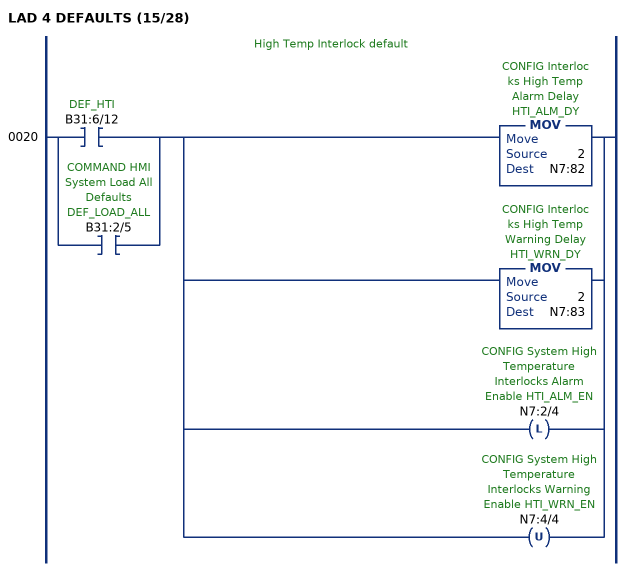
% Rung: 20 %
% High Temp Interlock default %
SOR BST XIC B31:6/12 NXB XIC B31:2/5 BND BST MOV 2 N7:82 NXB MOV 2 N7:83 NXB OTL N7:2/4 NXB OTU N7:4/4 BND EOR
%   B31:6/12  DEF_HTI %
%   B31:2/5  DEF_LOAD_ALL  "COMMAND HMI System Load All Defaults" %
%   N7:82  HTI_ALM_DY  "CONFIG Interlocks High Temp Alarm Delay" %
%   N7:83  HTI_WRN_DY  "CONFIG Interlocks High Temp Warning Delay" %
%   N7:2/4  HTI_ALM_EN  "CONFIG System High Temperature Interlocks Alarm Enable" %
%   N7:4/4  HTI_WRN_EN  "CONFIG System High Temperature Interlocks Warning Enable" %

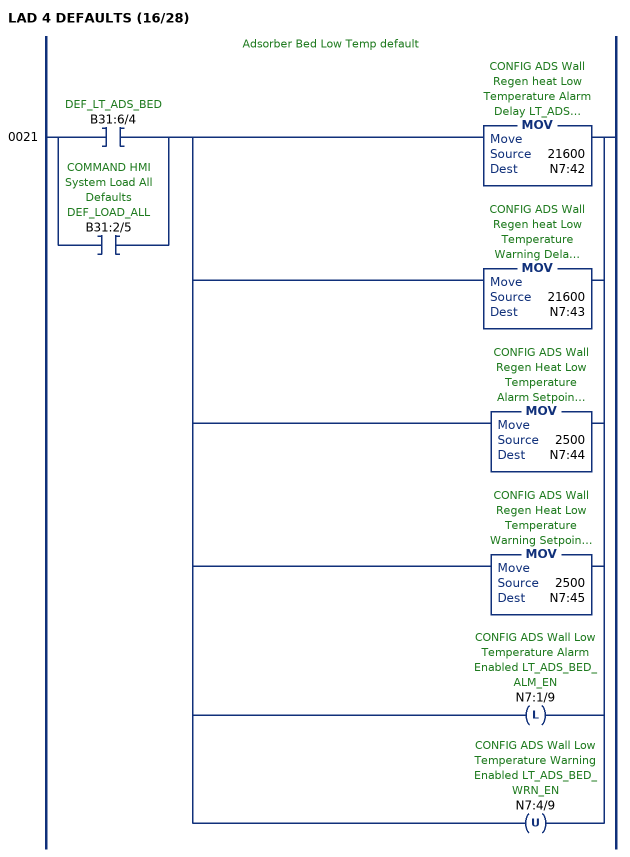
% Rung: 21 %
% Adsorber Bed Low Temp default %
SOR BST XIC B31:6/4 NXB XIC B31:2/5 BND BST MOV 21600 N7:42 NXB MOV 21600 N7:43 NXB MOV 2500 N7:44 NXB MOV 2500 N7:45 NXB OTL N7:1/9 NXB OTU N7:4/9 BND EOR
%   B31:6/4  DEF_LT_ADS_BED %
%   B31:2/5  DEF_LOAD_ALL  "COMMAND HMI System Load All Defaults" %
%   N7:42  LT_ADS_BED_ALM_DLY  "CONFIG ADS Wall Regen heat Low Temperature Alarm Delay" %
%   N7:43  LT_ADS_BED_WRN_DLY  "CONFIG ADS Wall Regen heat Low Temperature Warning Delay" %
%   N7:44  LT_ADS_BED_ALM_SP  "CONFIG ADS Wall Regen Heat Low Temperature Alarm Setpoint" %
%   N7:45  LT_ADS_BED_WRN_SP  "CONFIG ADS Wall Regen Heat Low Temperature Warning Setpoint" %
%   N7:1/9  LT_ADS_BED_ALM_EN  "CONFIG ADS Wall Low Temperature Alarm Enabled" %
%   N7:4/9  LT_ADS_BED_WRN_EN  "CONFIG ADS Wall Low Temperature Warning Enabled" %

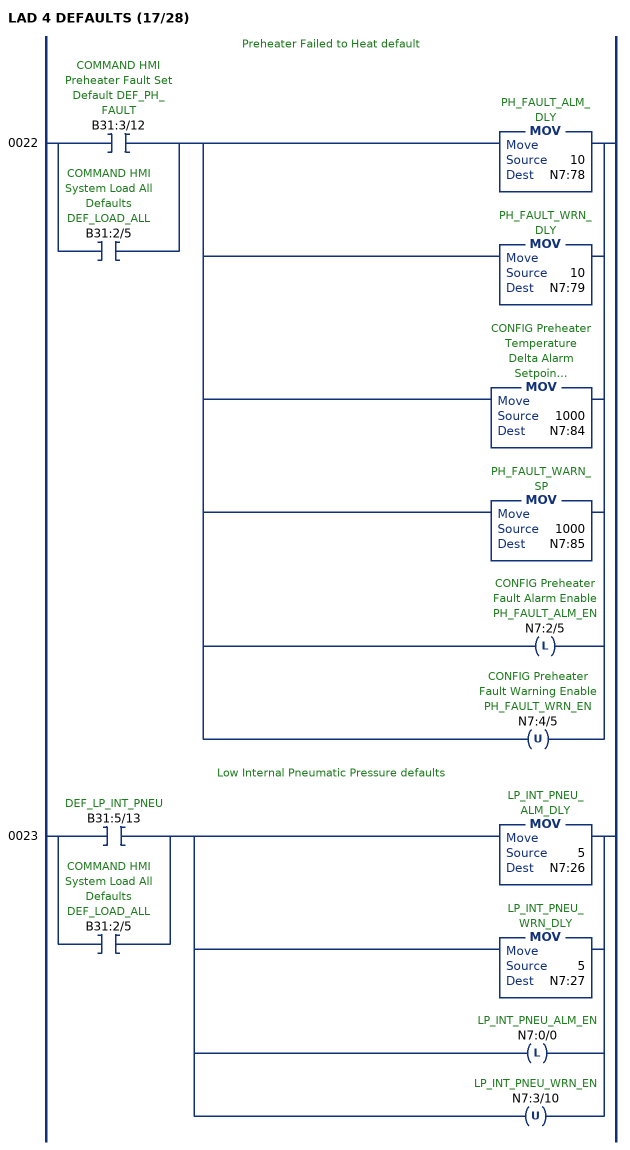
% Rung: 22 %
% Preheater Failed to Heat default %
SOR BST XIC B31:3/12 NXB XIC B31:2/5 BND BST MOV 10 N7:78 NXB MOV 10 N7:79 NXB MOV 1000 N7:84 NXB MOV 1000 N7:85 NXB OTL N7:2/5 NXB OTU N7:4/5 BND EOR
%   B31:3/12  DEF_PH_FAULT  "COMMAND HMI Preheater Fault Set Default" %
%   B31:2/5  DEF_LOAD_ALL  "COMMAND HMI System Load All Defaults" %
%   N7:78  PH_FAULT_ALM_DLY %
%   N7:79  PH_FAULT_WRN_DLY %
%   N7:84  PH_FAULT_ALARM_SP  "CONFIG Preheater Temperature Delta Alarm Setpoint" %
%   N7:85  PH_FAULT_WARN_SP %
%   N7:2/5  PH_FAULT_ALM_EN  "CONFIG Preheater Fault Alarm Enable" %
%   N7:4/5  PH_FAULT_WRN_EN  "CONFIG Preheater Fault Warning Enable" %
% Rung: 23 %
% Low Internal Pneumatic Pressure defaults %
SOR BST XIC B31:5/13 NXB XIC B31:2/5 BND BST MOV 5 N7:26 NXB MOV 5 N7:27 NXB OTL N7:0/0 NXB OTU N7:3/10 BND EOR
%   B31:5/13  DEF_LP_INT_PNEU %
%   B31:2/5  DEF_LOAD_ALL  "COMMAND HMI System Load All Defaults" %
%   N7:26  LP_INT_PNEU_ALM_DLY %
%   N7:27  LP_INT_PNEU_WRN_DLY %
%   N7:0/0  LP_INT_PNEU_ALM_EN %
%   N7:3/10  LP_INT_PNEU_WRN_EN %

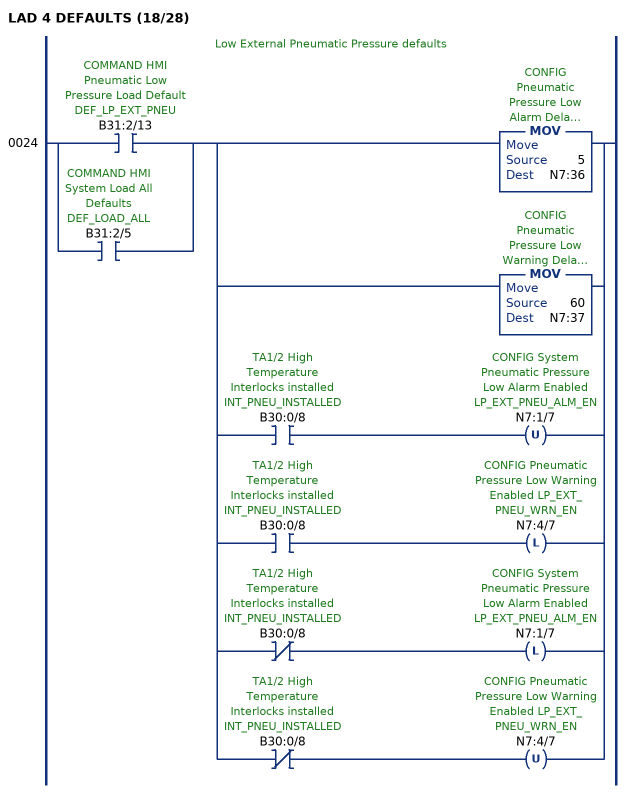
% Rung: 24 %
% Low External Pneumatic Pressure defaults %
SOR BST XIC B31:2/13 NXB XIC B31:2/5 BND BST MOV 5 N7:36 NXB MOV 60 N7:37 NXB XIC B30:0/8 OTU N7:1/7 NXB XIC B30:0/8 OTL N7:4/7 NXB XIO B30:0/8 OTL N7:1/7 NXB XIO B30:0/8 OTU N7:4/7 BND EOR
%   B31:2/13  DEF_LP_EXT_PNEU  "COMMAND HMI Pneumatic Low Pressure Load Default" %
%   B31:2/5  DEF_LOAD_ALL  "COMMAND HMI System Load All Defaults" %
%   N7:36  LP_EXT_PNEU_ALM_DLY  "CONFIG Pneumatic Pressure Low Alarm Delay" %
%   N7:37  LP_EXT_PNEU_WRN_DLY  "CONFIG Pneumatic Pressure Low Warning Delay" %
%   B30:0/8  INT_PNEU_INSTALLED  "TA1/2 High Temperature Interlocks installed" %
%   N7:1/7  LP_EXT_PNEU_ALM_EN  "CONFIG System Pneumatic Pressure Low Alarm Enabled" %
%   N7:4/7  LP_EXT_PNEU_WRN_EN  "CONFIG Pneumatic Pressure Low Warning Enabled" %

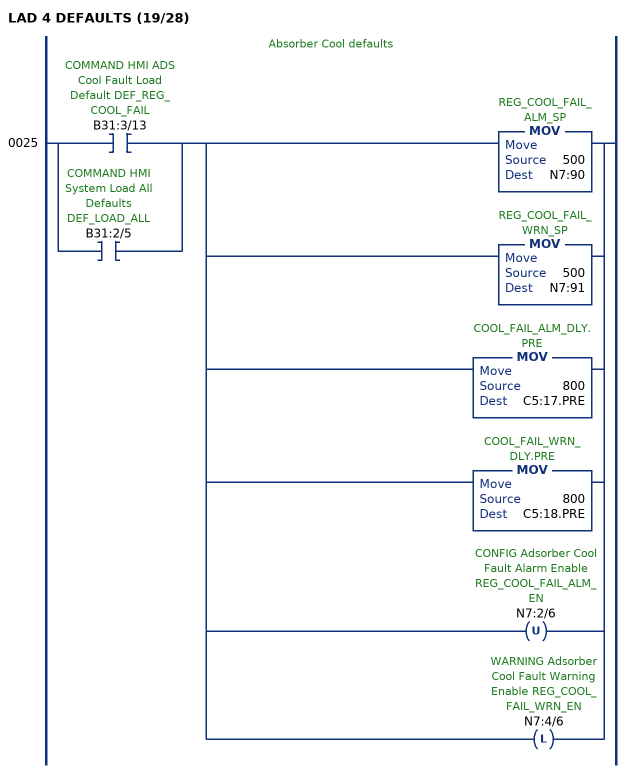
% Rung: 25 %
% Absorber Cool defaults %
SOR BST XIC B31:3/13 NXB XIC B31:2/5 BND BST MOV 500 N7:90 NXB MOV 500 N7:91 NXB MOV 800 C5:17.PRE NXB MOV 800 C5:18.PRE NXB OTU N7:2/6 NXB OTL N7:4/6 BND EOR
%   B31:3/13  DEF_REG_COOL_FAIL  "COMMAND HMI ADS Cool Fault Load Default" %
%   B31:2/5  DEF_LOAD_ALL  "COMMAND HMI System Load All Defaults" %
%   N7:90  REG_COOL_FAIL_ALM_SP %
%   N7:91  REG_COOL_FAIL_WRN_SP %
%   C5:17  COOL_FAIL_ALM_DLY %
%   C5:18  COOL_FAIL_WRN_DLY %
%   N7:2/6  REG_COOL_FAIL_ALM_EN  "CONFIG Adsorber Cool Fault Alarm Enable" %
%   N7:4/6  REG_COOL_FAIL_WRN_EN  "WARNING Adsorber Cool Fault Warning Enable" %

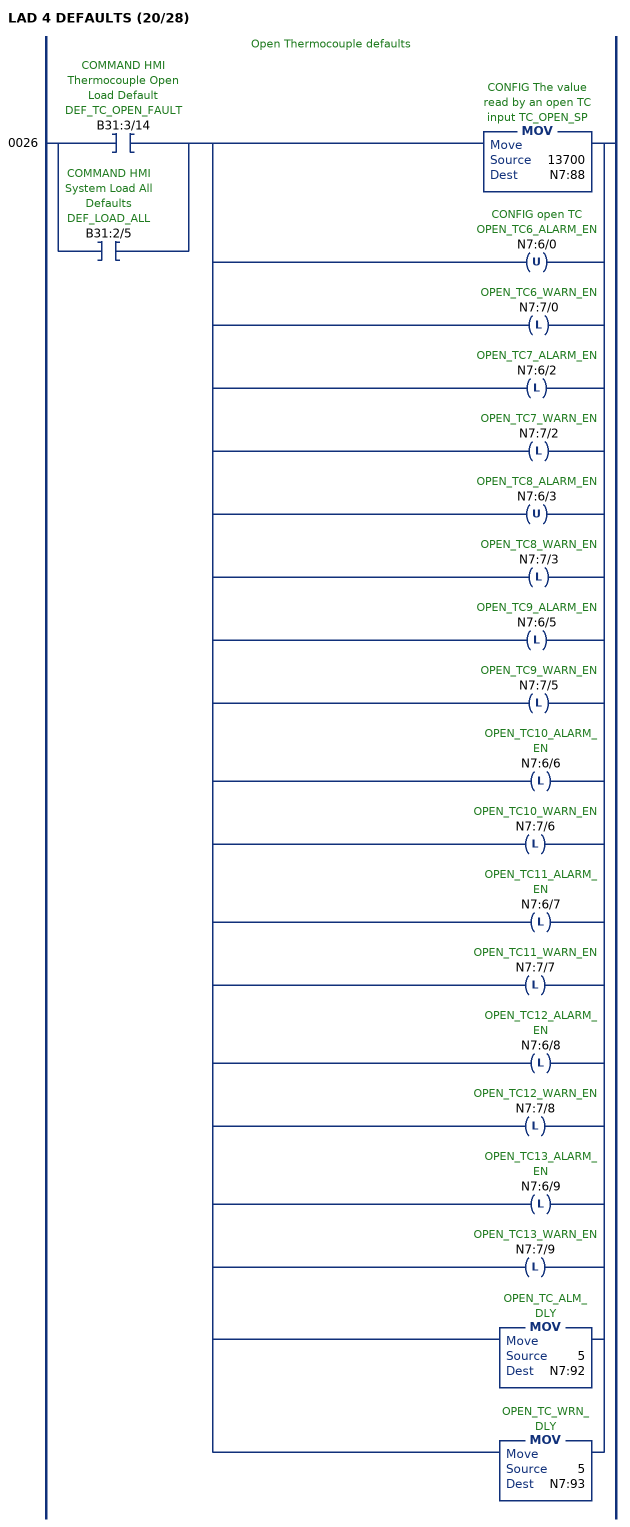
% Rung: 26 %
% Open Thermocouple defaults %
SOR BST XIC B31:3/14 NXB XIC B31:2/5 BND BST MOV 13700 N7:88 NXB OTU N7:6/0 NXB OTL N7:7/0 NXB OTL N7:6/2 NXB OTL N7:7/2 NXB OTU N7:6/3 NXB OTL N7:7/3 NXB OTL N7:6/5 NXB OTL N7:7/5 NXB OTL N7:6/6 NXB OTL N7:7/6 NXB OTL N7:6/7 NXB OTL N7:7/7 NXB OTL N7:6/8 NXB OTL N7:7/8 NXB OTL N7:6/9 NXB OTL N7:7/9 NXB MOV 5 N7:92 NXB MOV 5 N7:93 BND EOR
%   B31:3/14  DEF_TC_OPEN_FAULT  "COMMAND HMI Thermocouple Open Load Default" %
%   B31:2/5  DEF_LOAD_ALL  "COMMAND HMI System Load All Defaults" %
%   N7:88  TC_OPEN_SP  "CONFIG The value read by an open TC input" %
%   N7:6/0  OPEN_TC6_ALARM_EN  "CONFIG open TC" %
%   N7:7/0  OPEN_TC6_WARN_EN %
%   N7:6/2  OPEN_TC7_ALARM_EN %
%   N7:7/2  OPEN_TC7_WARN_EN %
%   N7:6/3  OPEN_TC8_ALARM_EN %
%   N7:7/3  OPEN_TC8_WARN_EN %
%   N7:6/5  OPEN_TC9_ALARM_EN %
%   N7:7/5  OPEN_TC9_WARN_EN %
%   N7:6/6  OPEN_TC10_ALARM_EN %
%   N7:7/6  OPEN_TC10_WARN_EN %
%   N7:6/7  OPEN_TC11_ALARM_EN %
%   N7:7/7  OPEN_TC11_WARN_EN %
%   N7:6/8  OPEN_TC12_ALARM_EN %
%   N7:7/8  OPEN_TC12_WARN_EN %
%   N7:6/9  OPEN_TC13_ALARM_EN %
%   N7:7/9  OPEN_TC13_WARN_EN %
%   N7:92  OPEN_TC_ALM_DLY %
%   N7:93  OPEN_TC_WRN_DLY %

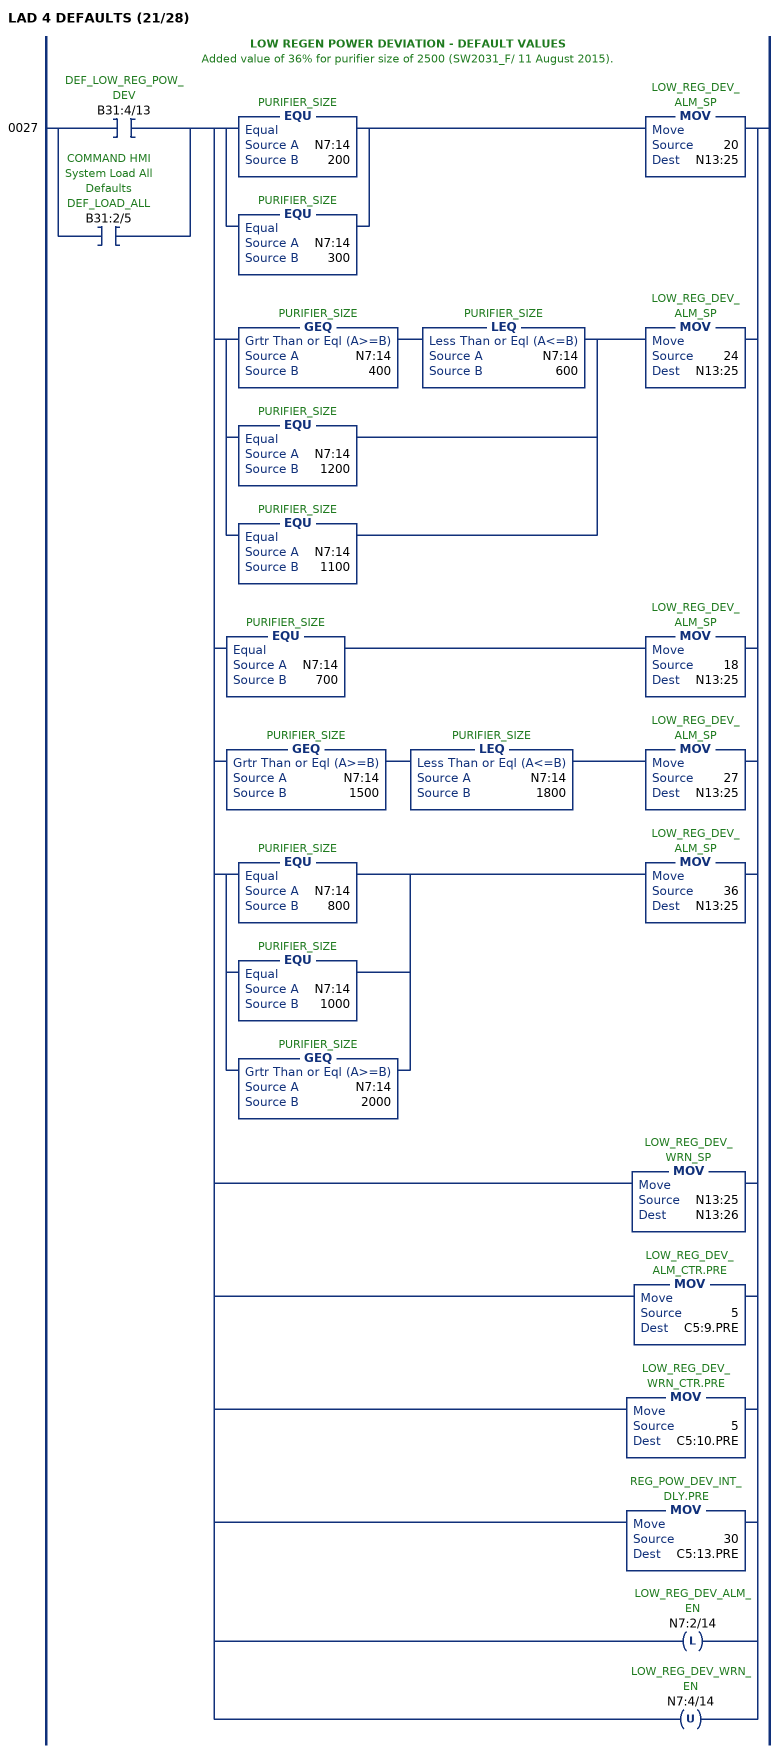
% Rung: 27 %
% TITLE: LOW REGEN POWER DEVIATION - DEFAULT VALUES %
% Added value of 36% for purifier size of 2500 (SW2031_F/ 11 August 2015). %
SOR BST XIC B31:4/13 NXB XIC B31:2/5 BND BST BST EQU N7:14 200 NXB EQU N7:14 300 BND MOV 20 N13:25 NXB BST GEQ N7:14 400 LEQ N7:14 600 NXB EQU N7:14 1200 NXB EQU N7:14 1100 BND MOV 24 N13:25 NXB EQU N7:14 700 MOV 18 N13:25 NXB GEQ N7:14 1500 LEQ N7:14 1800 MOV 27 N13:25 NXB BST EQU N7:14 800 NXB EQU N7:14 1000 NXB GEQ N7:14 2000 BND MOV 36 N13:25 NXB MOV N13:25 N13:26 NXB MOV 5 C5:9.PRE NXB MOV 5 C5:10.PRE NXB MOV 30 C5:13.PRE NXB OTL N7:2/14 NXB OTU N7:4/14 BND EOR
%   B31:4/13  DEF_LOW_REG_POW_DEV %
%   B31:2/5  DEF_LOAD_ALL  "COMMAND HMI System Load All Defaults" %
%   N7:14  PURIFIER_SIZE %
%   N13:25  LOW_REG_DEV_ALM_SP %
%   N13:26  LOW_REG_DEV_WRN_SP %
%   C5:9  LOW_REG_DEV_ALM_CTR %
%   C5:10  LOW_REG_DEV_WRN_CTR %
%   C5:13  REG_POW_DEV_INT_DLY %
%   N7:2/14  LOW_REG_DEV_ALM_EN %
%   N7:4/14  LOW_REG_DEV_WRN_EN %

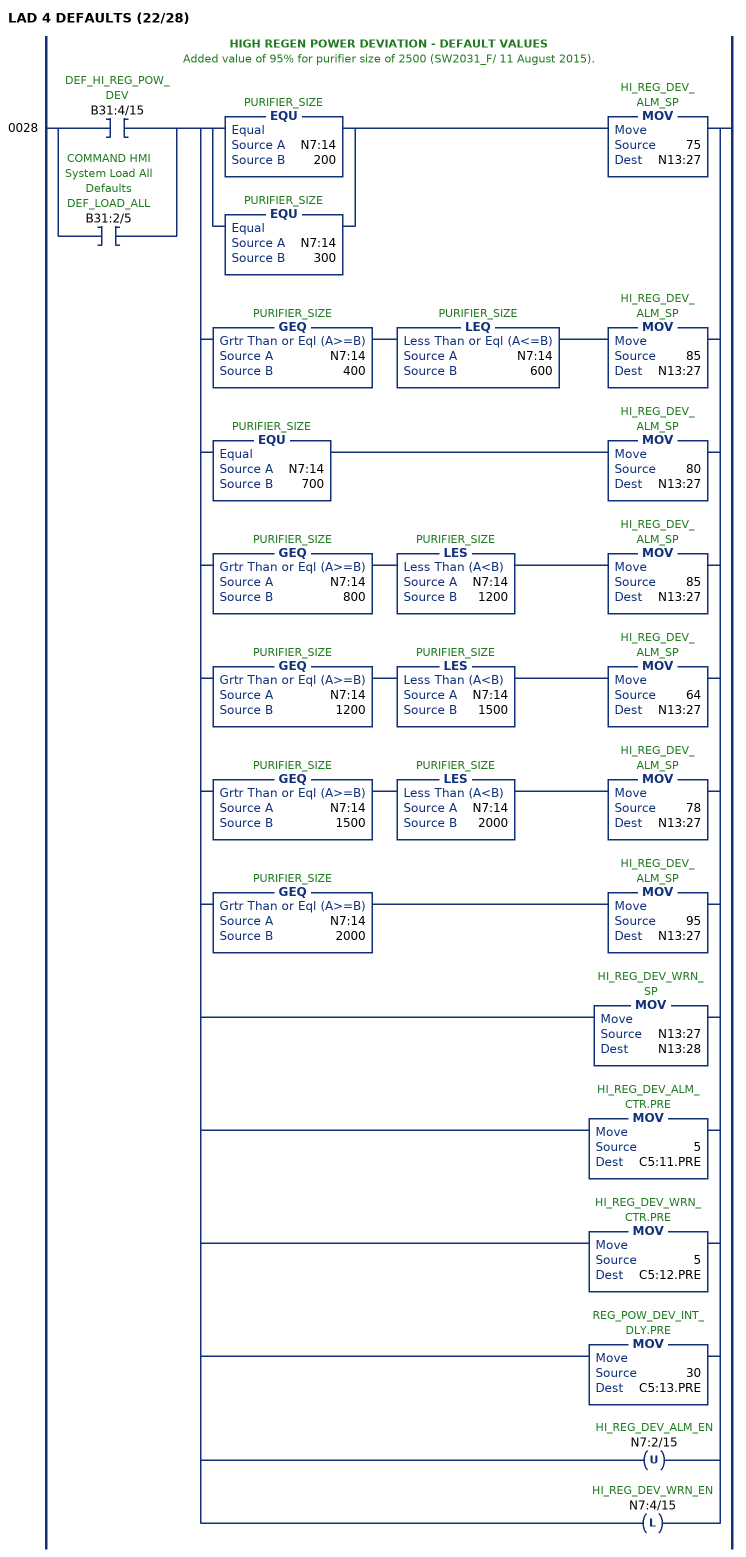
% Rung: 28 %
% TITLE: HIGH REGEN POWER DEVIATION - DEFAULT VALUES %
% Added value of 95% for purifier size of 2500 (SW2031_F/ 11 August 2015). %
SOR BST XIC B31:4/15 NXB XIC B31:2/5 BND BST BST EQU N7:14 200 NXB EQU N7:14 300 BND MOV 75 N13:27 NXB GEQ N7:14 400 LEQ N7:14 600 MOV 85 N13:27 NXB EQU N7:14 700 MOV 80 N13:27 NXB GEQ N7:14 800 LES N7:14 1200 MOV 85 N13:27 NXB GEQ N7:14 1200 LES N7:14 1500 MOV 64 N13:27 NXB GEQ N7:14 1500 LES N7:14 2000 MOV 78 N13:27 NXB GEQ N7:14 2000 MOV 95 N13:27 NXB MOV N13:27 N13:28 NXB MOV 5 C5:11.PRE NXB MOV 5 C5:12.PRE NXB MOV 30 C5:13.PRE NXB OTU N7:2/15 NXB OTL N7:4/15 BND EOR
%   B31:4/15  DEF_HI_REG_POW_DEV %
%   B31:2/5  DEF_LOAD_ALL  "COMMAND HMI System Load All Defaults" %
%   N7:14  PURIFIER_SIZE %
%   N13:27  HI_REG_DEV_ALM_SP %
%   N13:28  HI_REG_DEV_WRN_SP %
%   C5:11  HI_REG_DEV_ALM_CTR %
%   C5:12  HI_REG_DEV_WRN_CTR %
%   C5:13  REG_POW_DEV_INT_DLY %
%   N7:2/15  HI_REG_DEV_ALM_EN %
%   N7:4/15  HI_REG_DEV_WRN_EN %

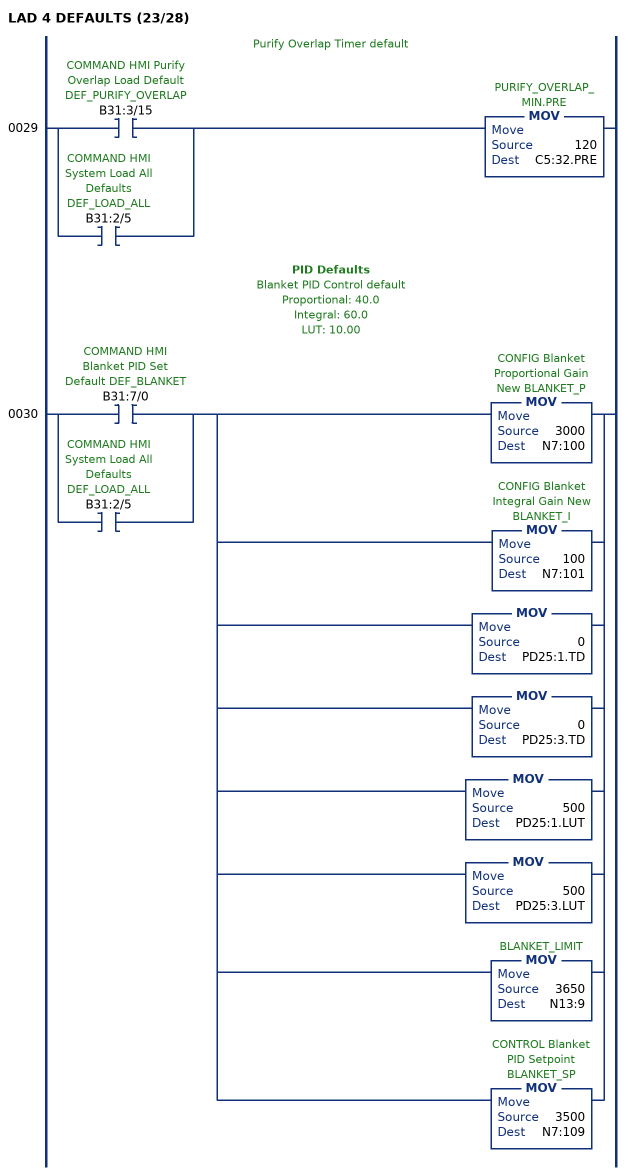
% Rung: 29 %
% Purify Overlap Timer default %
SOR BST XIC B31:3/15 NXB XIC B31:2/5 BND MOV 120 C5:32.PRE EOR
%   B31:3/15  DEF_PURIFY_OVERLAP  "COMMAND HMI Purify Overlap Load Default" %
%   B31:2/5  DEF_LOAD_ALL  "COMMAND HMI System Load All Defaults" %
%   C5:32  PURIFY_OVERLAP_MIN %
% Rung: 30 %
% TITLE: PID Defaults %
% Blanket PID Control default
% Proportional: 40.0
% Integral: 60.0
% LUT: 10.00 %
SOR BST XIC B31:7/0 NXB XIC B31:2/5 BND BST MOV 3000 N7:100 NXB MOV 100 N7:101 NXB MOV 0 PD25:1.TD NXB MOV 0 PD25:3.TD NXB MOV 500 PD25:1.LUT NXB MOV 500 PD25:3.LUT NXB MOV 3650 N13:9 NXB MOV 3500 N7:109 BND EOR
%   B31:7/0  DEF_BLANKET  "COMMAND HMI Blanket PID Set Default" %
%   B31:2/5  DEF_LOAD_ALL  "COMMAND HMI System Load All Defaults" %
%   N7:100  BLANKET_P  "CONFIG Blanket Proportional Gain New" %
%   N7:101  BLANKET_I  "CONFIG Blanket Integral Gain New" %
%   N13:9  BLANKET_LIMIT %
%   N7:109  BLANKET_SP  "CONTROL Blanket PID Setpoint" %

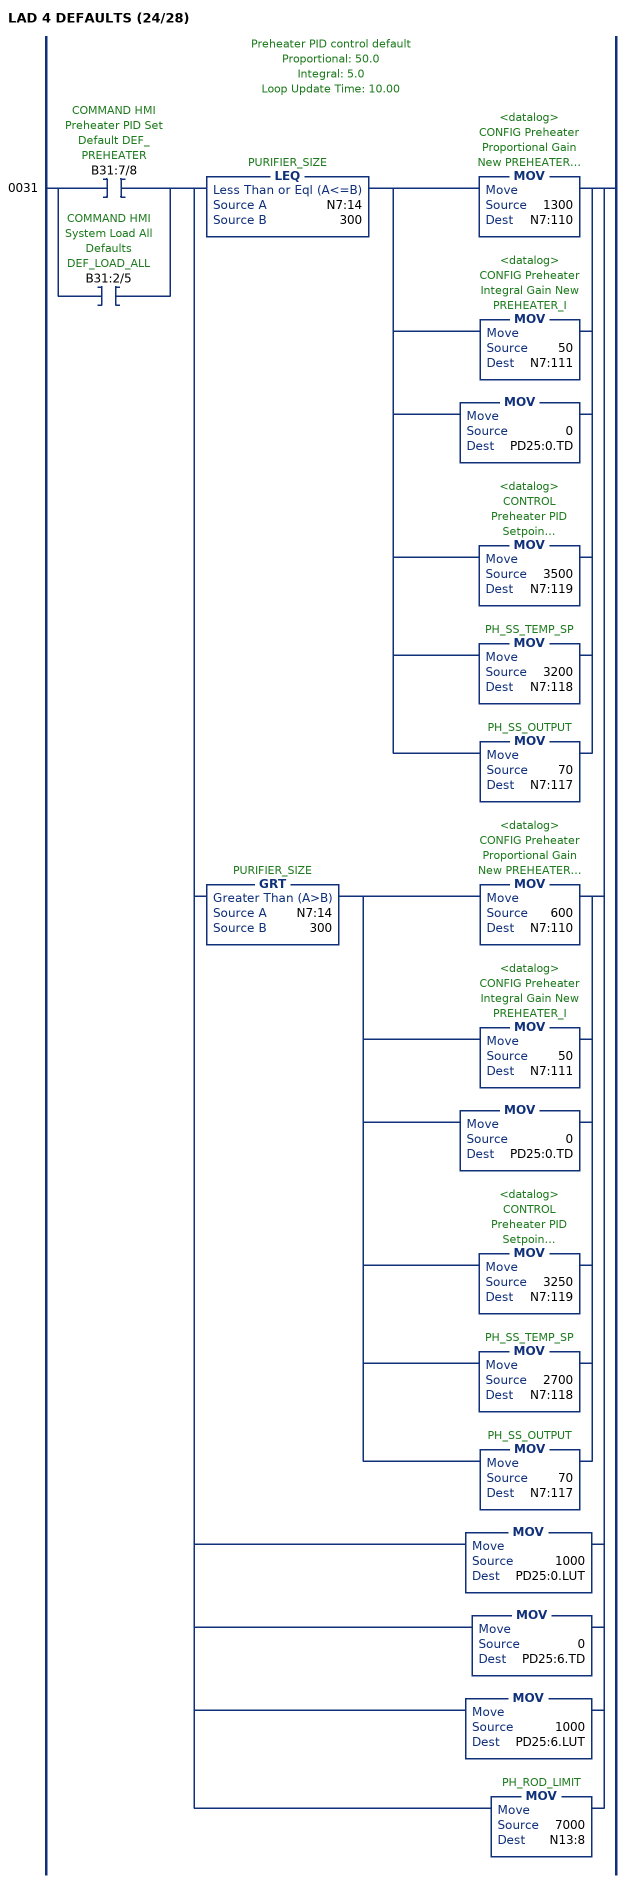
% Rung: 31 %
% Preheater PID control default
% Proportional: 50.0
% Integral: 5.0
% Loop Update Time: 10.00 %
SOR BST XIC B31:7/8 NXB XIC B31:2/5 BND BST LEQ N7:14 300 BST MOV 1300 N7:110 NXB MOV 50 N7:111 NXB MOV 0 PD25:0.TD NXB MOV 3500 N7:119 NXB MOV 3200 N7:118 NXB MOV 70 N7:117 BND NXB GRT N7:14 300 BST MOV 600 N7:110 NXB MOV 50 N7:111 NXB MOV 0 PD25:0.TD NXB MOV 3250 N7:119 NXB MOV 2700 N7:118 NXB MOV 70 N7:117 BND NXB MOV 1000 PD25:0.LUT NXB MOV 0 PD25:6.TD NXB MOV 1000 PD25:6.LUT NXB MOV 7000 N13:8 BND EOR
%   B31:7/8  DEF_PREHEATER  "COMMAND HMI Preheater PID Set Default" %
%   B31:2/5  DEF_LOAD_ALL  "COMMAND HMI System Load All Defaults" %
%   N7:14  PURIFIER_SIZE %
%   N7:110  PREHEATER_P  "<datalog> CONFIG Preheater Proportional Gain New" %
%   N7:111  PREHEATER_I  "<datalog> CONFIG Preheater Integral Gain New" %
%   N7:119  PREHEATER_SP  "<datalog> CONTROL Preheater PID Setpoint" %
%   N7:118  PH_SS_TEMP_SP %
%   N7:117  PH_SS_OUTPUT %
%   N13:8  PH_ROD_LIMIT %

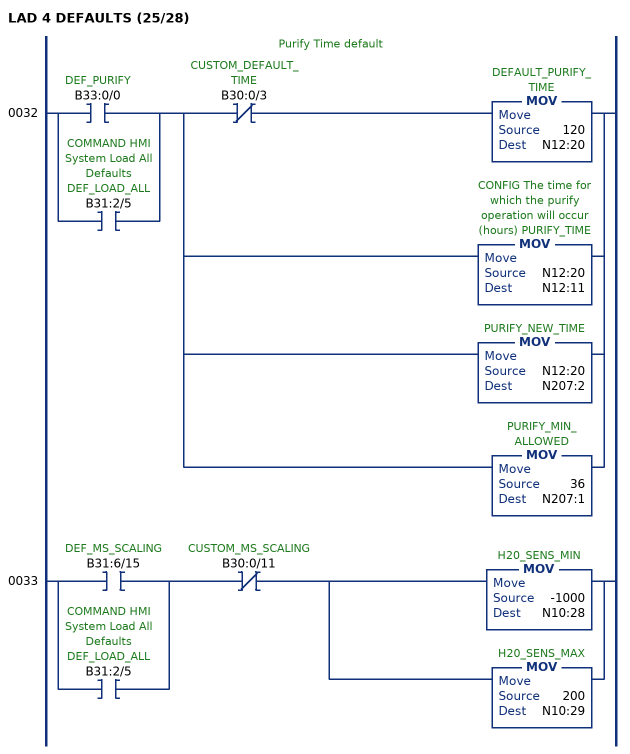
% Rung: 32 %
% Purify Time default %
SOR BST XIC B33:0/0 NXB XIC B31:2/5 BND BST XIO B30:0/3 MOV 120 N12:20 NXB MOV N12:20 N12:11 NXB MOV N12:20 N207:2 NXB MOV 36 N207:1 BND EOR
%   B33:0/0  DEF_PURIFY %
%   B31:2/5  DEF_LOAD_ALL  "COMMAND HMI System Load All Defaults" %
%   B30:0/3  CUSTOM_DEFAULT_TIME %
%   N12:20  DEFAULT_PURIFY_TIME %
%   N12:11  PURIFY_TIME  "CONFIG The time for which the purify operation will occur (hours)" %
%   N207:2  PURIFY_NEW_TIME %
%   N207:1  PURIFY_MIN_ALLOWED %
% Rung: 33 %
SOR BST XIC B31:6/15 NXB XIC B31:2/5 BND XIO B30:0/11 BST MOV -1000 N10:28 NXB MOV 200 N10:29 BND EOR
%   B31:6/15  DEF_MS_SCALING %
%   B31:2/5  DEF_LOAD_ALL  "COMMAND HMI System Load All Defaults" %
%   B30:0/11  CUSTOM_MS_SCALING %
%   N10:28  H20_SENS_MIN %
%   N10:29  H20_SENS_MAX %

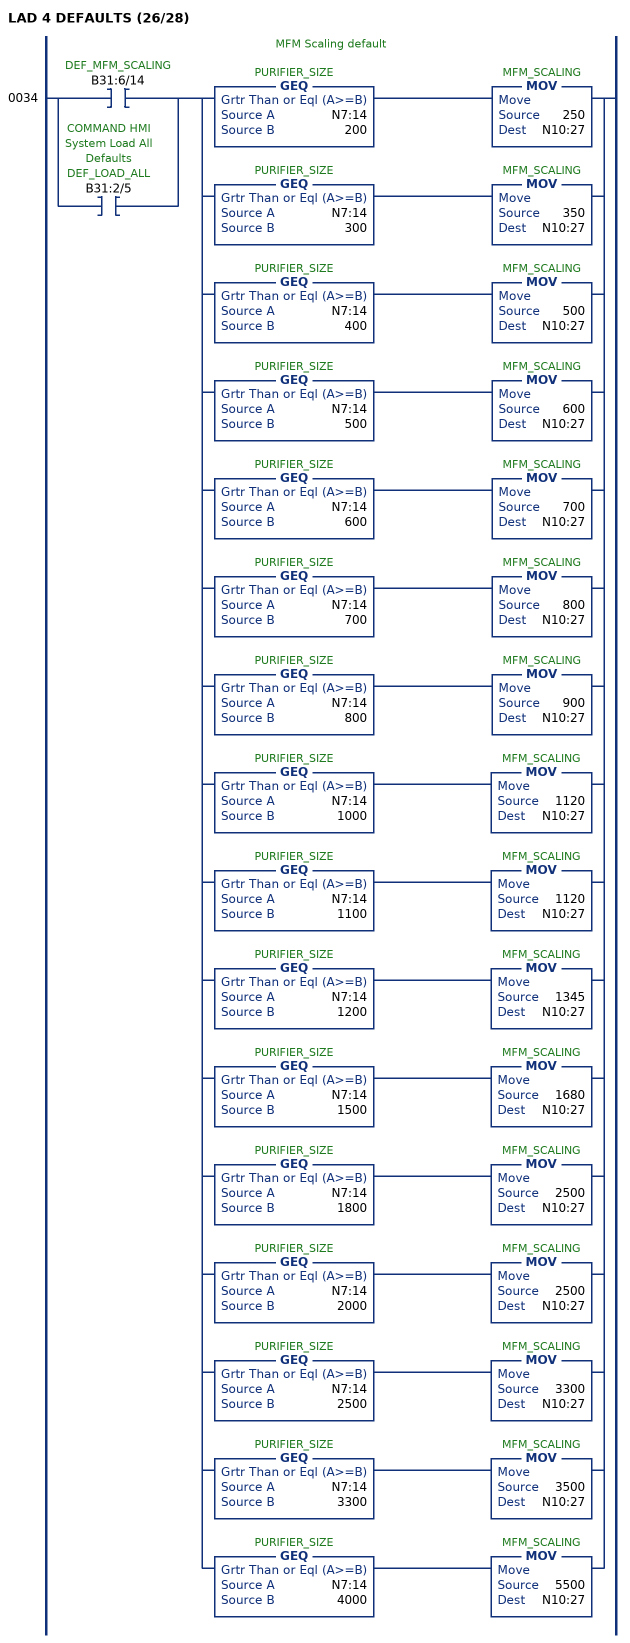
% Rung: 34 %
% MFM Scaling default %
SOR BST XIC B31:6/14 NXB XIC B31:2/5 BND BST GEQ N7:14 200 MOV 250 N10:27 NXB GEQ N7:14 300 MOV 350 N10:27 NXB GEQ N7:14 400 MOV 500 N10:27 NXB GEQ N7:14 500 MOV 600 N10:27 NXB GEQ N7:14 600 MOV 700 N10:27 NXB GEQ N7:14 700 MOV 800 N10:27 NXB GEQ N7:14 800 MOV 900 N10:27 NXB GEQ N7:14 1000 MOV 1120 N10:27 NXB GEQ N7:14 1100 MOV 1120 N10:27 NXB GEQ N7:14 1200 MOV 1345 N10:27 NXB GEQ N7:14 1500 MOV 1680 N10:27 NXB GEQ N7:14 1800 MOV 2500 N10:27 NXB GEQ N7:14 2000 MOV 2500 N10:27 NXB GEQ N7:14 2500 MOV 3300 N10:27 NXB GEQ N7:14 3300 MOV 3500 N10:27 NXB GEQ N7:14 4000 MOV 5500 N10:27 BND EOR
%   B31:6/14  DEF_MFM_SCALING %
%   B31:2/5  DEF_LOAD_ALL  "COMMAND HMI System Load All Defaults" %
%   N7:14  PURIFIER_SIZE %
%   N10:27  MFM_SCALING %

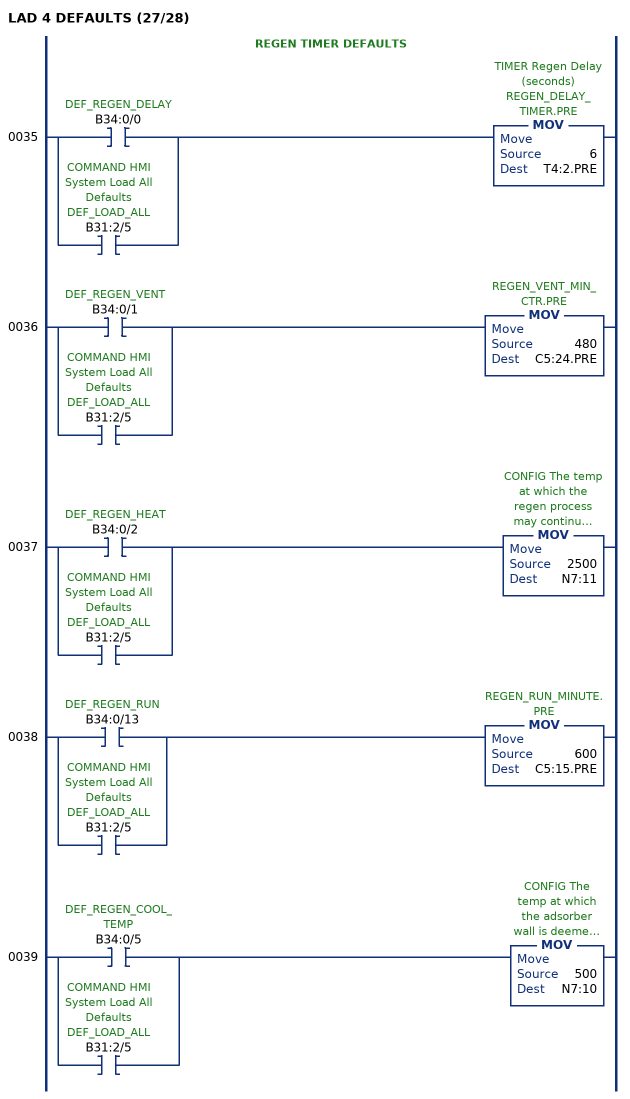
% Rung: 35 %
% TITLE: REGEN TIMER DEFAULTS %
SOR BST XIC B34:0/0 NXB XIC B31:2/5 BND MOV 6 T4:2.PRE EOR
%   B34:0/0  DEF_REGEN_DELAY %
%   B31:2/5  DEF_LOAD_ALL  "COMMAND HMI System Load All Defaults" %
%   T4:2  REGEN_DELAY_TIMER  "TIMER Regen Delay (seconds)" %
% Rung: 36 %
SOR BST XIC B34:0/1 NXB XIC B31:2/5 BND MOV 480 C5:24.PRE EOR
%   B34:0/1  DEF_REGEN_VENT %
%   B31:2/5  DEF_LOAD_ALL  "COMMAND HMI System Load All Defaults" %
%   C5:24  REGEN_VENT_MIN_CTR %
% Rung: 37 %
SOR BST XIC B34:0/2 NXB XIC B31:2/5 BND MOV 2500 N7:11 EOR
%   B34:0/2  DEF_REGEN_HEAT %
%   B31:2/5  DEF_LOAD_ALL  "COMMAND HMI System Load All Defaults" %
%   N7:11  ADS_BED_TEMP_HIGH  "CONFIG The temp at which the regen process may continue" %
% Rung: 38 %
SOR BST XIC B34:0/13 NXB XIC B31:2/5 BND MOV 600 C5:15.PRE EOR
%   B34:0/13  DEF_REGEN_RUN %
%   B31:2/5  DEF_LOAD_ALL  "COMMAND HMI System Load All Defaults" %
%   C5:15  REGEN_RUN_MINUTE %
% Rung: 39 %
SOR BST XIC B34:0/5 NXB XIC B31:2/5 BND MOV 500 N7:10 EOR
%   B34:0/5  DEF_REGEN_COOL_TEMP %
%   B31:2/5  DEF_LOAD_ALL  "COMMAND HMI System Load All Defaults" %
%   N7:10  ADS_WALL_TEMP_COOL  "CONFIG The temp at which the adsorber wall is deemed to be cool enough to purify" %

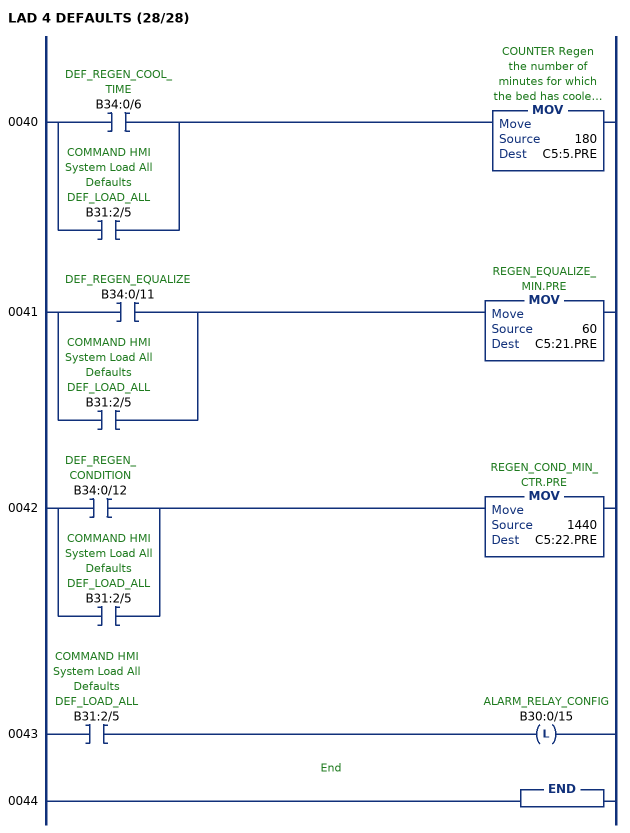
% Rung: 40 %
SOR BST XIC B34:0/6 NXB XIC B31:2/5 BND MOV 180 C5:5.PRE EOR
%   B34:0/6  DEF_REGEN_COOL_TIME %
%   B31:2/5  DEF_LOAD_ALL  "COMMAND HMI System Load All Defaults" %
%   C5:5  REGEN_COOL_MINUTE  "COUNTER Regen the number of minutes for which the bed has cooled" %
% Rung: 41 %
SOR BST XIC B34:0/11 NXB XIC B31:2/5 BND MOV 60 C5:21.PRE EOR
%   B34:0/11  DEF_REGEN_EQUALIZE %
%   B31:2/5  DEF_LOAD_ALL  "COMMAND HMI System Load All Defaults" %
%   C5:21  REGEN_EQUALIZE_MIN %
% Rung: 42 %
SOR BST XIC B34:0/12 NXB XIC B31:2/5 BND MOV 1440 C5:22.PRE EOR
%   B34:0/12  DEF_REGEN_CONDITION %
%   B31:2/5  DEF_LOAD_ALL  "COMMAND HMI System Load All Defaults" %
%   C5:22  REGEN_COND_MIN_CTR %
% Rung: 43 %
SOR XIC B31:2/5 OTL B30:0/15 EOR
%   B31:2/5  DEF_LOAD_ALL  "COMMAND HMI System Load All Defaults" %
%   B30:0/15  ALARM_RELAY_CONFIG %
% Rung: 44 %
% End %
SOR END EOR

LADDER 5 "SYS_FAULTS"    % Monitors the system fault conditions %
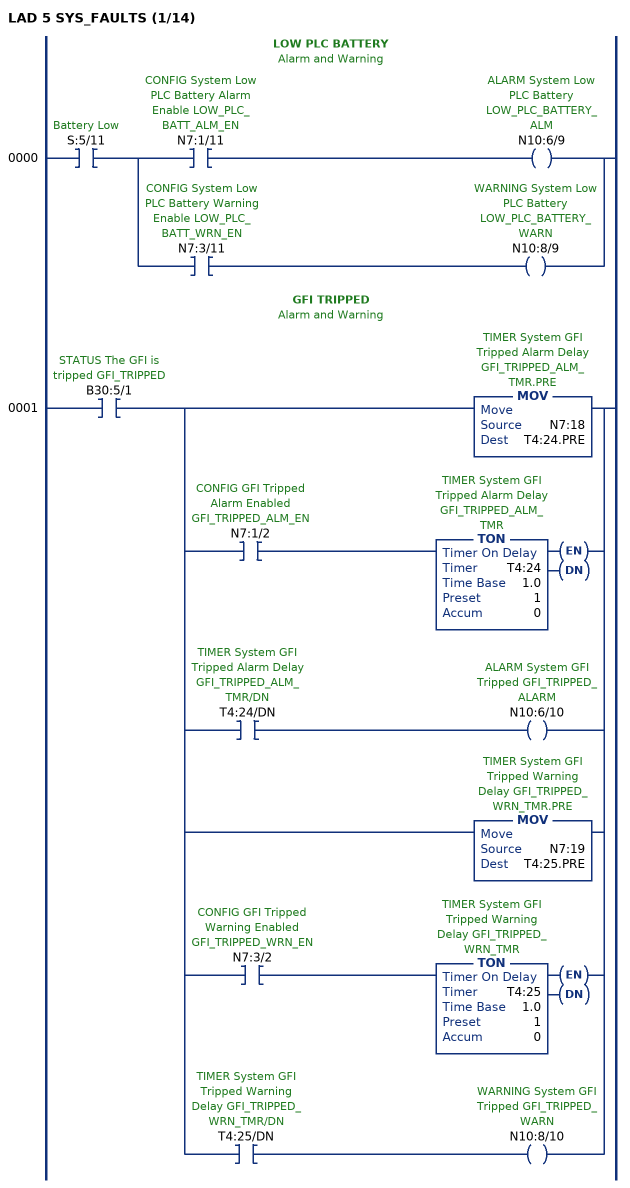
% Rung: 0 %
% TITLE: LOW PLC BATTERY %
% Alarm and Warning %
SOR XIC S:5/11 BST XIC N7:1/11 OTE N10:6/9 NXB XIC N7:3/11 OTE N10:8/9 BND EOR
%   S:5/11  "Battery Low" %
%   N7:1/11  LOW_PLC_BATT_ALM_EN  "CONFIG System Low PLC Battery Alarm Enable" %
%   N10:6/9  LOW_PLC_BATTERY_ALM  "ALARM System Low PLC Battery" %
%   N7:3/11  LOW_PLC_BATT_WRN_EN  "CONFIG System Low PLC Battery Warning Enable" %
%   N10:8/9  LOW_PLC_BATTERY_WARN  "WARNING System Low PLC Battery" %
% Rung: 1 %
% TITLE: GFI TRIPPED %
% Alarm and Warning %
SOR XIC B30:5/1 BST MOV N7:18 T4:24.PRE NXB XIC N7:1/2 TON T4:24 1.0 1 0 NXB XIC T4:24/DN OTE N10:6/10 NXB MOV N7:19 T4:25.PRE NXB XIC N7:3/2 TON T4:25 1.0 1 0 NXB XIC T4:25/DN OTE N10:8/10 BND EOR
%   B30:5/1  GFI_TRIPPED  "STATUS The GFI is tripped" %
%   N7:18  GFI_TRIPPED_ALM_DLY  "CONFIG GFI fault alarm delay" %
%   T4:24  GFI_TRIPPED_ALM_TMR  "TIMER System GFI Tripped Alarm Delay" %
%   N7:1/2  GFI_TRIPPED_ALM_EN  "CONFIG GFI Tripped Alarm Enabled" %
%   N10:6/10  GFI_TRIPPED_ALARM  "ALARM System GFI Tripped" %
%   N7:19  GFI_TRIPPED_WRN_DLY  "CONFIG GFI fault warning delay" %
%   T4:25  GFI_TRIPPED_WRN_TMR  "TIMER System GFI Tripped Warning Delay" %
%   N7:3/2  GFI_TRIPPED_WRN_EN  "CONFIG GFI Tripped Warning Enabled" %
%   N10:8/10  GFI_TRIPPED_WARN  "WARNING System GFI Tripped" %

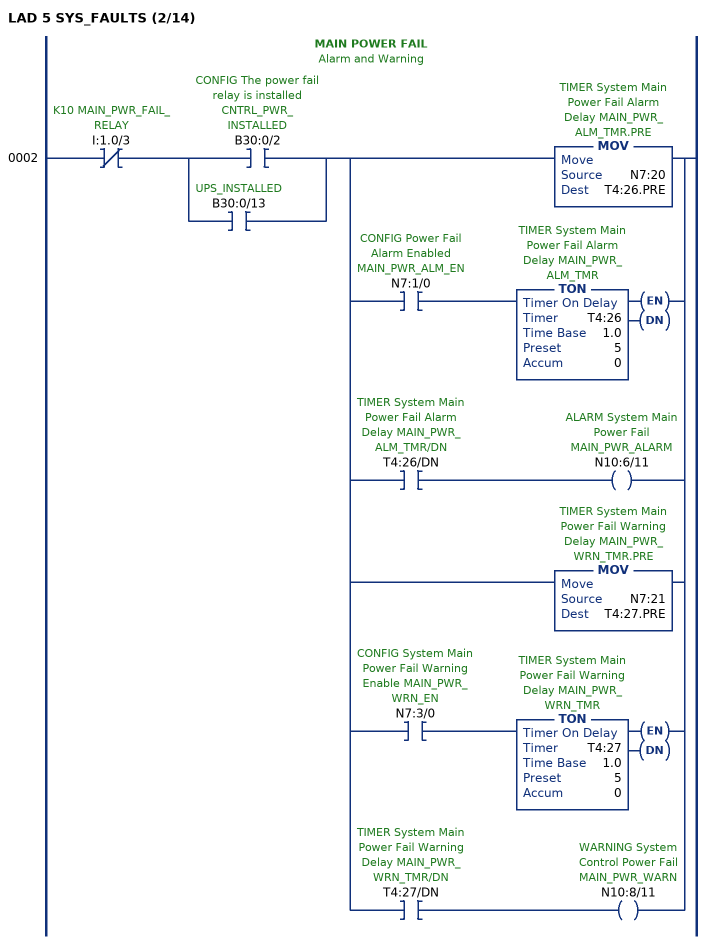
% Rung: 2 %
% TITLE: MAIN POWER FAIL %
% Alarm and Warning %
SOR XIO I:1.0/3 BST XIC B30:0/2 NXB XIC B30:0/13 BND BST MOV N7:20 T4:26.PRE NXB XIC N7:1/0 TON T4:26 1.0 5 0 NXB XIC T4:26/DN OTE N10:6/11 NXB MOV N7:21 T4:27.PRE NXB XIC N7:3/0 TON T4:27 1.0 5 0 NXB XIC T4:27/DN OTE N10:8/11 BND EOR
%   I:1.0/3  MAIN_PWR_FAIL_RELAY  "K10" %
%   B30:0/2  CNTRL_PWR_INSTALLED  "CONFIG The power fail relay is installed" %
%   B30:0/13  UPS_INSTALLED %
%   N7:20  PWR_FAIL_ALM_DELAY  "CONFIG System Power failure Alarm Delay" %
%   T4:26  MAIN_PWR_ALM_TMR  "TIMER System Main Power Fail Alarm Delay" %
%   N7:1/0  MAIN_PWR_ALM_EN  "CONFIG Power Fail Alarm Enabled" %
%   N10:6/11  MAIN_PWR_ALARM  "ALARM System Main Power Fail" %
%   N7:21  PWR_FAIL_WRN_DELAY  "CONFIG System Power Failure Warning Delay" %
%   T4:27  MAIN_PWR_WRN_TMR  "TIMER System Main Power Fail Warning Delay" %
%   N7:3/0  MAIN_PWR_WRN_EN  "CONFIG System Main Power Fail Warning Enable" %
%   N10:8/11  MAIN_PWR_WARN  "WARNING System Control Power Fail" %

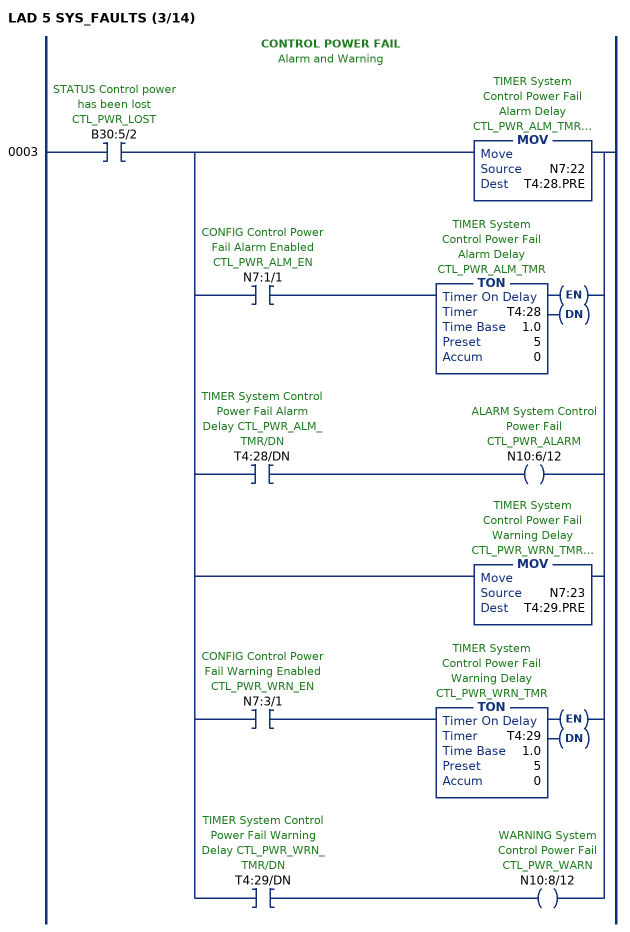
% Rung: 3 %
% TITLE: CONTROL POWER FAIL %
% Alarm and Warning %
SOR XIC B30:5/2 BST MOV N7:22 T4:28.PRE NXB XIC N7:1/1 TON T4:28 1.0 5 0 NXB XIC T4:28/DN OTE N10:6/12 NXB MOV N7:23 T4:29.PRE NXB XIC N7:3/1 TON T4:29 1.0 5 0 NXB XIC T4:29/DN OTE N10:8/12 BND EOR
%   B30:5/2  CTL_PWR_LOST  "STATUS Control power has been lost" %
%   N7:22  CTL_PWR_FAIL_ALM_DLY  "CONFIG Control power alarm delay setpoint" %
%   T4:28  CTL_PWR_ALM_TMR  "TIMER System Control Power Fail Alarm Delay" %
%   N7:1/1  CTL_PWR_ALM_EN  "CONFIG Control Power Fail Alarm Enabled" %
%   N10:6/12  CTL_PWR_ALARM  "ALARM System Control Power Fail" %
%   N7:23  CTL_PWR_FAIL_WRN_DLY  "CONFIG Control power failure warning delay setpoint" %
%   T4:29  CTL_PWR_WRN_TMR  "TIMER System Control Power Fail Warning Delay" %
%   N7:3/1  CTL_PWR_WRN_EN  "CONFIG Control Power Fail Warning Enabled" %
%   N10:8/12  CTL_PWR_WARN  "WARNING System Control Power Fail" %

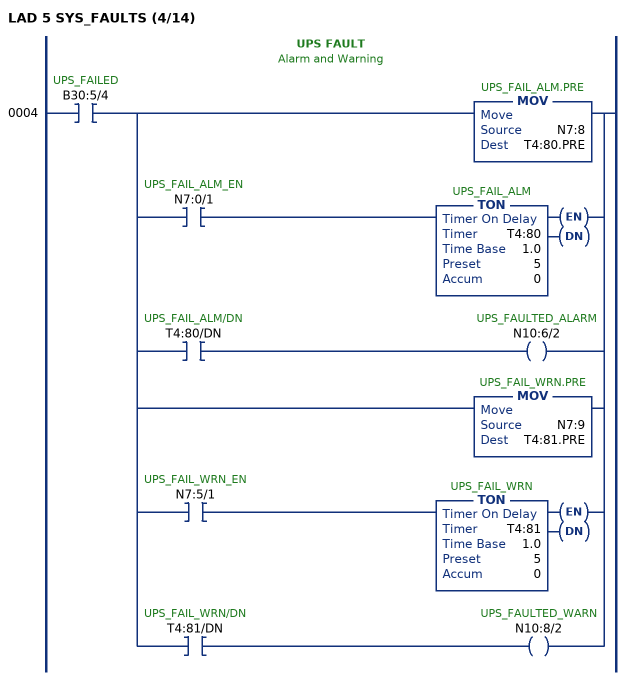
% Rung: 4 %
% TITLE: UPS FAULT %
% Alarm and Warning %
SOR XIC B30:5/4 BST MOV N7:8 T4:80.PRE NXB XIC N7:0/1 TON T4:80 1.0 5 0 NXB XIC T4:80/DN OTE N10:6/2 NXB MOV N7:9 T4:81.PRE NXB XIC N7:5/1 TON T4:81 1.0 5 0 NXB XIC T4:81/DN OTE N10:8/2 BND EOR
%   B30:5/4  UPS_FAILED %
%   N7:8  UPS_FAIL_ALM_DLY %
%   T4:80  UPS_FAIL_ALM %
%   N7:0/1  UPS_FAIL_ALM_EN %
%   N10:6/2  UPS_FAULTED_ALARM %
%   N7:9  UPS_FAIL_WRN_DLY %
%   T4:81  UPS_FAIL_WRN %
%   N7:5/1  UPS_FAIL_WRN_EN %
%   N10:8/2  UPS_FAULTED_WARN %

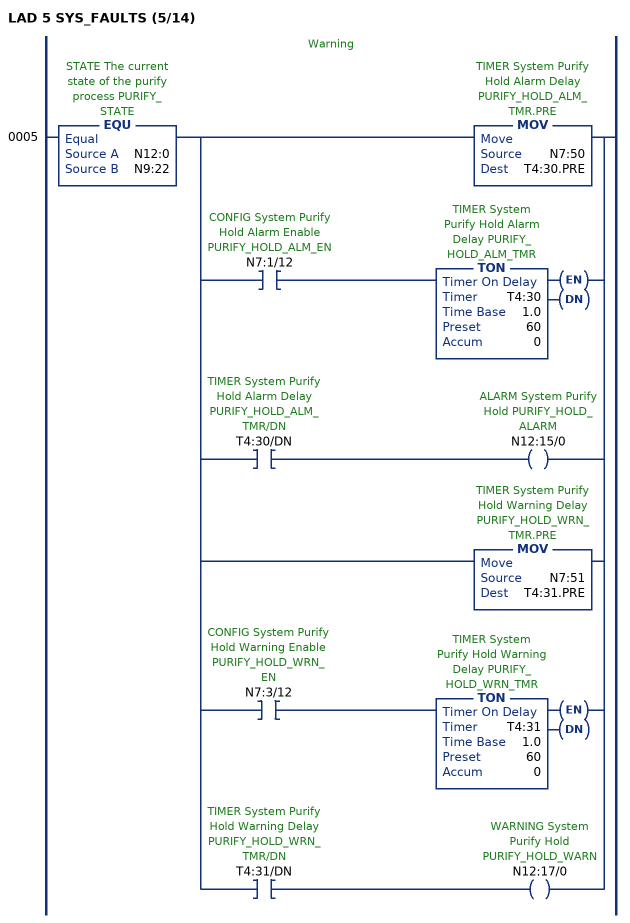
% Rung: 5 %
% Warning %
SOR EQU N12:0 N9:22 BST MOV N7:50 T4:30.PRE NXB XIC N7:1/12 TON T4:30 1.0 60 0 NXB XIC T4:30/DN OTE N12:15/0 NXB MOV N7:51 T4:31.PRE NXB XIC N7:3/12 TON T4:31 1.0 60 0 NXB XIC T4:31/DN OTE N12:17/0 BND EOR
%   N12:0  PURIFY_STATE  "STATE The current state of the purify process" %
%   N9:22  PURIFY_HOLD  "STATE Purify Hold" %
%   N7:50  PURIFY_HOLD_ALM_DLY  "CONFIG System Purify Hold Alarm Delay" %
%   T4:30  PURIFY_HOLD_ALM_TMR  "TIMER System Purify Hold Alarm Delay" %
%   N7:1/12  PURIFY_HOLD_ALM_EN  "CONFIG System Purify Hold Alarm Enable" %
%   N12:15/0  PURIFY_HOLD_ALARM  "ALARM System Purify Hold" %
%   N7:51  PURIFY_HOLD_WRN_DLY  "CONFIG System Purify Hold Warning Delay" %
%   T4:31  PURIFY_HOLD_WRN_TMR  "TIMER System Purify Hold Warning Delay" %
%   N7:3/12  PURIFY_HOLD_WRN_EN  "CONFIG System Purify Hold Warning Enable" %
%   N12:17/0  PURIFY_HOLD_WARN  "WARNING System Purify Hold" %

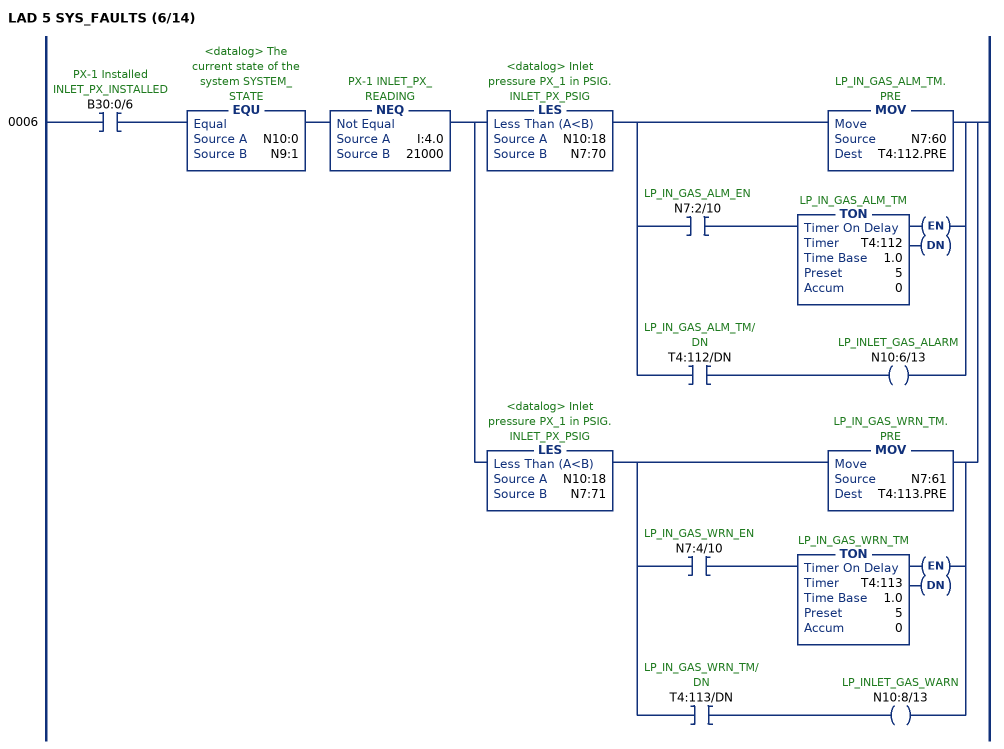
% Rung: 6 %
SOR XIC B30:0/6 EQU N10:0 N9:1 NEQ I:4.0 21000 BST LES N10:18 N7:70 BST MOV N7:60 T4:112.PRE NXB XIC N7:2/10 TON T4:112 1.0 5 0 NXB XIC T4:112/DN OTE N10:6/13 BND NXB LES N10:18 N7:71 BST MOV N7:61 T4:113.PRE NXB XIC N7:4/10 TON T4:113 1.0 5 0 NXB XIC T4:113/DN OTE N10:8/13 BND BND EOR
%   B30:0/6  INLET_PX_INSTALLED  "PX-1 Installed" %
%   N10:0  SYSTEM_STATE  "<datalog> The current state of the system" %
%   N9:1  SYSTEM_PROCESS  "STATE System Process" %
%   I:4.0  INLET_PX_READING  "PX-1" %
%   N10:18  INLET_PX_PSIG  "<datalog> Inlet pressure PX_1 in PSIG." %
%   N7:70  LP_IN_GAS_ALM_SP %
%   N7:60  LP_GAS_ALM_DLY  "CONFIG System Low Gas Pressure Alarm Delay" %
%   T4:112  LP_IN_GAS_ALM_TM %
%   N7:2/10  LP_IN_GAS_ALM_EN %
%   N10:6/13  LP_INLET_GAS_ALARM %
%   N7:71  LP_IN_GAS_WRN_SP %
%   N7:61  LP_GAS_WRN_DLY  "CONFIG System Low Gas Pressure Warning Delay" %
%   T4:113  LP_IN_GAS_WRN_TM %
%   N7:4/10  LP_IN_GAS_WRN_EN %
%   N10:8/13  LP_INLET_GAS_WARN %

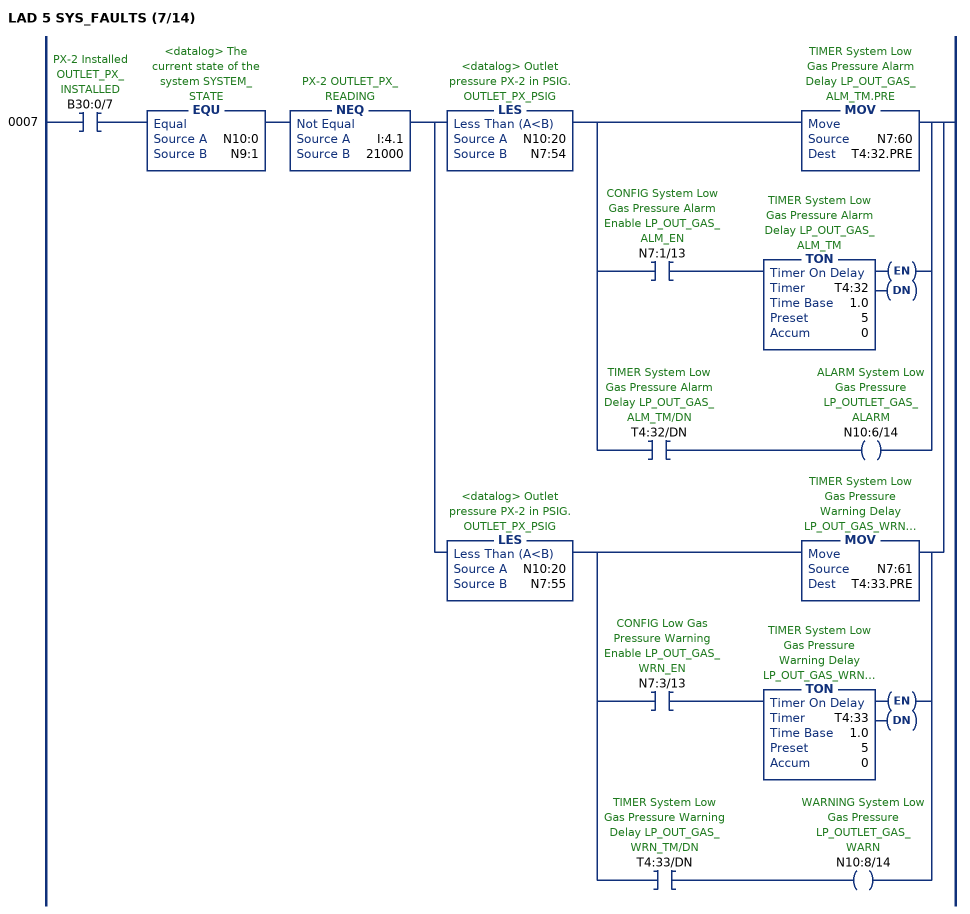
% Rung: 7 %
SOR XIC B30:0/7 EQU N10:0 N9:1 NEQ I:4.1 21000 BST LES N10:20 N7:54 BST MOV N7:60 T4:32.PRE NXB XIC N7:1/13 TON T4:32 1.0 5 0 NXB XIC T4:32/DN OTE N10:6/14 BND NXB LES N10:20 N7:55 BST MOV N7:61 T4:33.PRE NXB XIC N7:3/13 TON T4:33 1.0 5 0 NXB XIC T4:33/DN OTE N10:8/14 BND BND EOR
%   B30:0/7  OUTLET_PX_INSTALLED  "PX-2 Installed" %
%   N10:0  SYSTEM_STATE  "<datalog> The current state of the system" %
%   N9:1  SYSTEM_PROCESS  "STATE System Process" %
%   I:4.1  OUTLET_PX_READING  "PX-2" %
%   N10:20  OUTLET_PX_PSIG  "<datalog> Outlet pressure PX-2 in PSIG." %
%   N7:54  LP_OUT_GAS_ALM_SP  "CONFIG System Gas Inlet Pressure Low Alarm Setpoint" %
%   N7:60  LP_GAS_ALM_DLY  "CONFIG System Low Gas Pressure Alarm Delay" %
%   T4:32  LP_OUT_GAS_ALM_TM  "TIMER System Low Gas Pressure Alarm Delay" %
%   N7:1/13  LP_OUT_GAS_ALM_EN  "CONFIG System Low Gas Pressure Alarm Enable" %
%   N10:6/14  LP_OUTLET_GAS_ALARM  "ALARM System Low Gas Pressure" %
%   N7:55  LP_OUT_GAS_WRN_SP  "CONFIG System Gas Inlet Pressure Low Warning Setpoint" %
%   N7:61  LP_GAS_WRN_DLY  "CONFIG System Low Gas Pressure Warning Delay" %
%   T4:33  LP_OUT_GAS_WRN_TM  "TIMER System Low Gas Pressure Warning Delay" %
%   N7:3/13  LP_OUT_GAS_WRN_EN  "CONFIG Low Gas Pressure Warning Enable" %
%   N10:8/14  LP_OUTLET_GAS_WARN  "WARNING System Low Gas Pressure" %

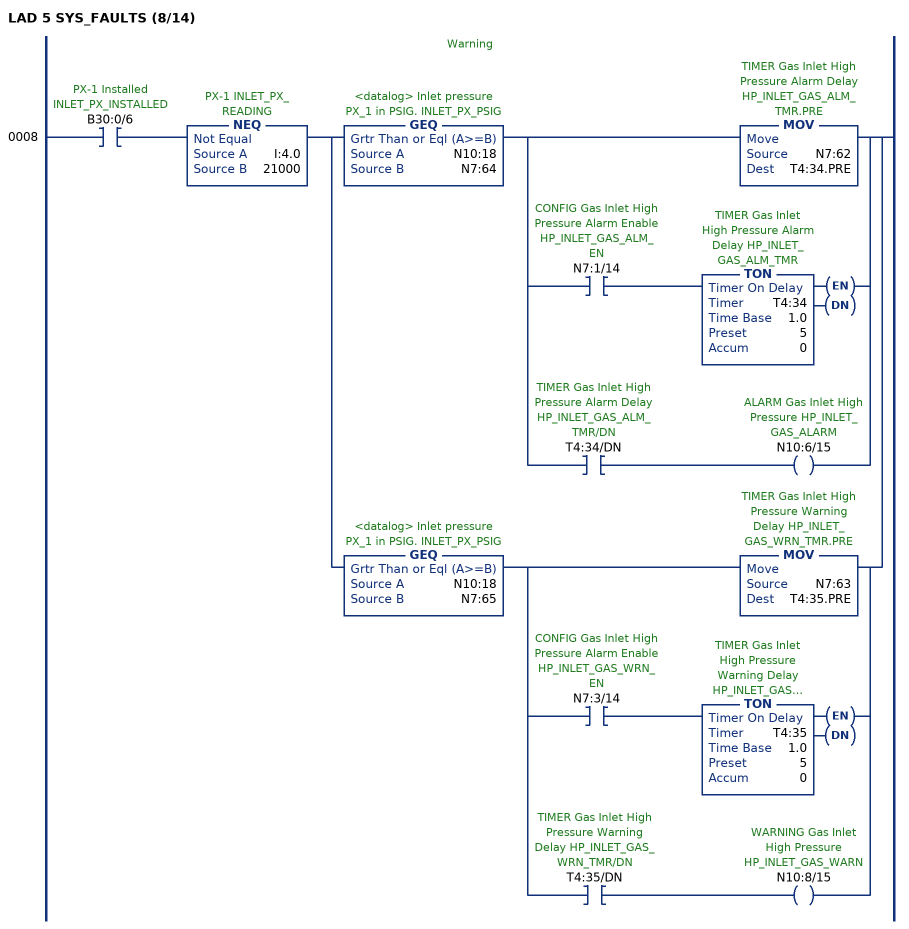
% Rung: 8 %
% Warning %
SOR XIC B30:0/6 NEQ I:4.0 21000 BST GEQ N10:18 N7:64 BST MOV N7:62 T4:34.PRE NXB XIC N7:1/14 TON T4:34 1.0 5 0 NXB XIC T4:34/DN OTE N10:6/15 BND NXB GEQ N10:18 N7:65 BST MOV N7:63 T4:35.PRE NXB XIC N7:3/14 TON T4:35 1.0 5 0 NXB XIC T4:35/DN OTE N10:8/15 BND BND EOR
%   B30:0/6  INLET_PX_INSTALLED  "PX-1 Installed" %
%   I:4.0  INLET_PX_READING  "PX-1" %
%   N10:18  INLET_PX_PSIG  "<datalog> Inlet pressure PX_1 in PSIG." %
%   N7:64  HP_INLET_GAS_ALM_SP  "CONFIG Gas Inlet High Pressure Alarm Setpoint" %
%   N7:62  HP_INLET_GAS_ALM_DLY  "CONFIG Gas Inlet High Pressure Alarm Delay" %
%   T4:34  HP_INLET_GAS_ALM_TMR  "TIMER Gas Inlet High Pressure Alarm Delay" %
%   N7:1/14  HP_INLET_GAS_ALM_EN  "CONFIG Gas Inlet High Pressure Alarm Enable" %
%   N10:6/15  HP_INLET_GAS_ALARM  "ALARM Gas Inlet High Pressure" %
%   N7:65  HP_INLET_GAS_WRN_SP  "CONFIG Gas Inlet High Pressure Warning Setpoint" %
%   N7:63  HP_INLET_GAS_WRN_DLY  "CONFIG Gas Inlet High Pressure Warning Delay" %
%   T4:35  HP_INLET_GAS_WRN_TMR  "TIMER Gas Inlet High Pressure Warning Delay" %
%   N7:3/14  HP_INLET_GAS_WRN_EN  "CONFIG Gas Inlet High Pressure Alarm Enable" %
%   N10:8/15  HP_INLET_GAS_WARN  "WARNING Gas Inlet High Pressure" %

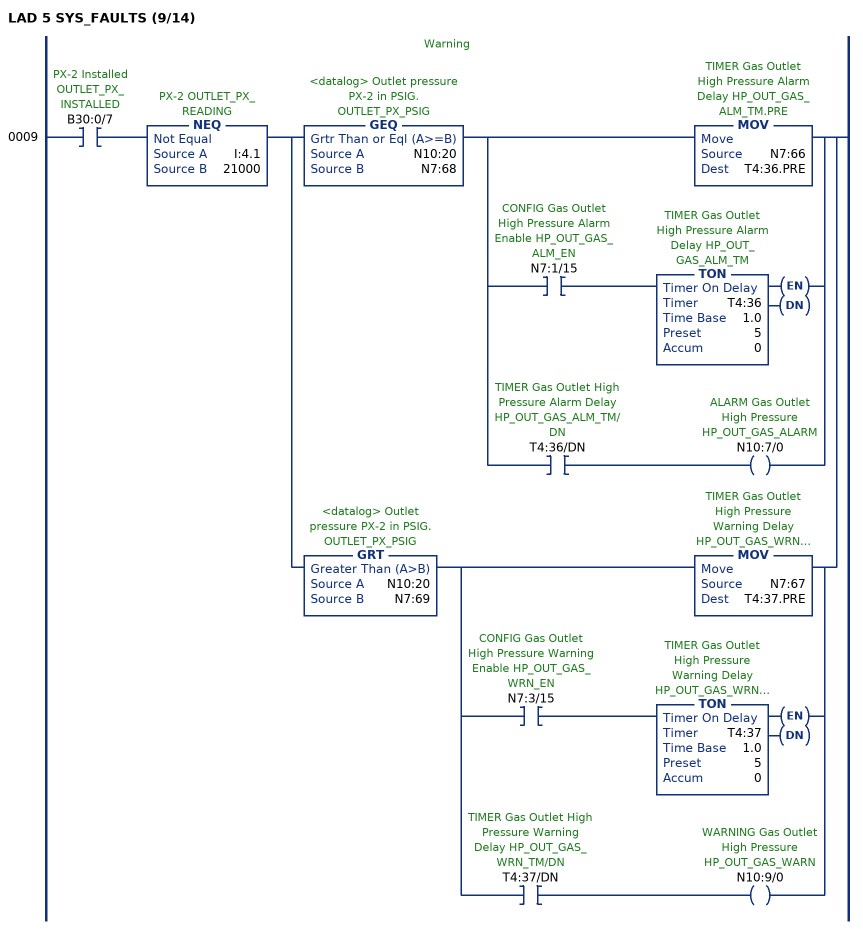
% Rung: 9 %
% Warning %
SOR XIC B30:0/7 NEQ I:4.1 21000 BST GEQ N10:20 N7:68 BST MOV N7:66 T4:36.PRE NXB XIC N7:1/15 TON T4:36 1.0 5 0 NXB XIC T4:36/DN OTE N10:7/0 BND NXB GRT N10:20 N7:69 BST MOV N7:67 T4:37.PRE NXB XIC N7:3/15 TON T4:37 1.0 5 0 NXB XIC T4:37/DN OTE N10:9/0 BND BND EOR
%   B30:0/7  OUTLET_PX_INSTALLED  "PX-2 Installed" %
%   I:4.1  OUTLET_PX_READING  "PX-2" %
%   N10:20  OUTLET_PX_PSIG  "<datalog> Outlet pressure PX-2 in PSIG." %
%   N7:68  HP_OUT_GAS_ALM_SP  "CONFIG Gas Outlet High Pressure Alarm Setpoint" %
%   N7:66  HP_OUT_GAS_ALM_DLY  "CONFIG Gas Outlet High Pressure Alarm Deley" %
%   T4:36  HP_OUT_GAS_ALM_TM  "TIMER Gas Outlet High Pressure Alarm Delay" %
%   N7:1/15  HP_OUT_GAS_ALM_EN  "CONFIG Gas Outlet High Pressure Alarm Enable" %
%   N10:7/0  HP_OUT_GAS_ALARM  "ALARM Gas Outlet High Pressure" %
%   N7:69  HP_OUT_GAS_WRN_SP  "CONFIG Gas Outlet High Pressure Warning Setpoint" %
%   N7:67  HP_OUT_GAS_WRN_DLY  "CONFIG Gas Outlet High Pressure Warning Delay" %
%   T4:37  HP_OUT_GAS_WRN_TM  "TIMER Gas Outlet High Pressure Warning Delay" %
%   N7:3/15  HP_OUT_GAS_WRN_EN  "CONFIG Gas Outlet High Pressure Warning Enable" %
%   N10:9/0  HP_OUT_GAS_WARN  "WARNING Gas Outlet High Pressure" %

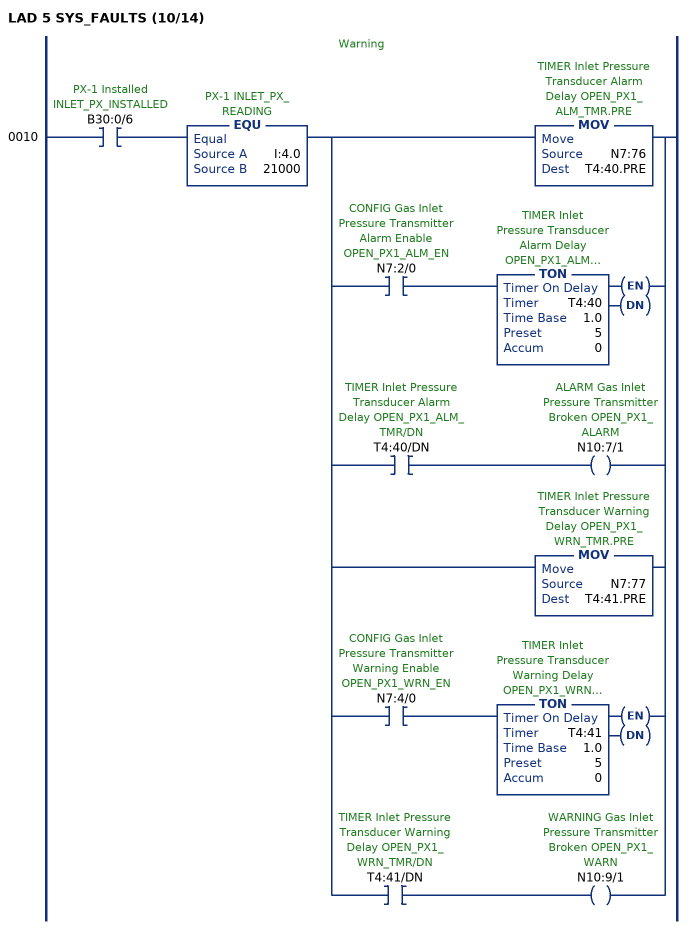
% Rung: 10 %
% Warning %
SOR XIC B30:0/6 EQU I:4.0 21000 BST MOV N7:76 T4:40.PRE NXB XIC N7:2/0 TON T4:40 1.0 5 0 NXB XIC T4:40/DN OTE N10:7/1 NXB MOV N7:77 T4:41.PRE NXB XIC N7:4/0 TON T4:41 1.0 5 0 NXB XIC T4:41/DN OTE N10:9/1 BND EOR
%   B30:0/6  INLET_PX_INSTALLED  "PX-1 Installed" %
%   I:4.0  INLET_PX_READING  "PX-1" %
%   N7:76  OPEN_PX1_ALM_DLY  "CONFIG Gas Inlet Pressure Transducer Alarm Delay" %
%   T4:40  OPEN_PX1_ALM_TMR  "TIMER Inlet Pressure Transducer Alarm Delay" %
%   N7:2/0  OPEN_PX1_ALM_EN  "CONFIG Gas Inlet Pressure Transmitter Alarm Enable" %
%   N10:7/1  OPEN_PX1_ALARM  "ALARM Gas Inlet Pressure Transmitter Broken" %
%   N7:77  OPEN_PX1_WRN_DLY  "CONFIG Gas Inlet Pressure Transducer Warning Delay" %
%   T4:41  OPEN_PX1_WRN_TMR  "TIMER Inlet Pressure Transducer Warning Delay" %
%   N7:4/0  OPEN_PX1_WRN_EN  "CONFIG Gas Inlet Pressure Transmitter Warning Enable" %
%   N10:9/1  OPEN_PX1_WARN  "WARNING Gas Inlet Pressure Transmitter Broken" %

